Universal Robots URScript: UR10-test.urscript

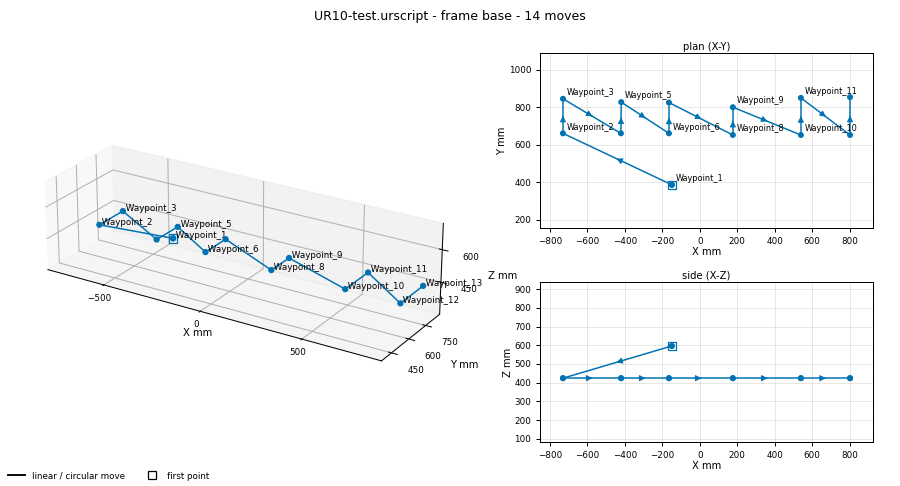
[picture p0: tool path of UR10-test.urscript in frame base, 14 of 14 moves have a stored position in this frame; points joined in program order, loops and branches not executed]
global Waypoint_1_p=p[-.148623716255, .387020693657, .596263904947, 2.224016818754, -2.218863100459, .000000000047]
global Waypoint_1_q=[-1.6361330038861635, -2.1105279423675096, 2.098508978739188, -1.5587831056934593, -1.5658103921715565, 1.5027728108834797]
global Waypoint_2_p=p[-.729817873873, .661722231264, .424287796426, -2.218887695886, 2.218882381559, -.005675531927]
global Waypoint_2_q=[-0.9138925478017441, -1.0490834600145664, 1.3516796273042528, -1.8702687876866584, -1.569889898709345, 2.2296846505934624]
global Waypoint_3_p=p[-.729817873828, .846264544764, .424287796402, -2.218887695886, 2.218882381560, -.005675531928]
global Waypoint_3_q=[-1.0153653607439015, -0.8157632596228916, 0.9656489876250722, -1.7179844037908198, -1.5701368644487452, 2.1274887333166923]
global Waypoint_4_p=p[-.420560802575, .661722231064, .424287796370, -2.218887695885, 2.218882381559, -.005675531928]
global Waypoint_4_q=[-1.2279537001817111, -1.3629806130695812, 1.794165965681119, -2.0002576570402937, -1.5708128857489623, 1.9161374014142538]
global Waypoint_5_p=p[-.418875864551, .828377650801, .424287796356, -2.218887695885, 2.218882381559, -.005675531928]
global Waypoint_5_q=[-1.2908790378613233, -1.1397118299440727, 1.489741921074341, -1.9194085745795313, -1.5708031426775904, 1.8529114400786177]
global Waypoint_6_p=p[-.164110914671, .661722231020, .424287796367, -2.218887695885, 2.218882381559, -.005675531929]
global Waypoint_6_q=[-1.5850637794811266, -1.5267522206750428, 1.9827905031090738, -2.026900558052507, -1.5711626782692507, 1.5590634072767182]
global Waypoint_7_p=p[-.164110914672, .826173042611, .424287796333, -2.218887695885, 2.218882381559, -.005675531929]
global Waypoint_7_q=[-1.582343695273308, -1.2729320930252044, 1.678075854753021, -1.9759921143142556, -1.5710752378853288, 1.5616684247757715]
global Waypoint_8_p=p[.177031398866, .652910761193, .424287796275, -2.218887695885, 2.218882381559, -.005675531929]
global Waypoint_8_q=[-2.0951142953865762, -1.535769708009413, 1.9928181636409832, -2.030398815561191, -1.5704868658568802, 1.049019558354602]
global Waypoint_9_p=p[.177031398835, .801253074719, .424287796241, -2.218887695885, 2.218882381559, -.005675531929]
global Waypoint_9_q=[-2.0015173847793495, -1.306690370177332, 1.7232682354739524, -1.9895026104403168, -1.5706322771175376, 1.1425409229913175]
global Waypoint_10_p=p[.540139343172, .652910760996, .424287796193, -2.218887695885, 2.218882381559, -.005675531929]
global Waypoint_10_q=[-2.4686027585240176, -1.2655837432115984, 1.6690811447534415, -1.9782898517891594, -1.5691603256432396, 0.6754183849426623]
global Waypoint_11_p=p[.540139343077, .850906857836, .424287796146, -2.218887695885, 2.218882381559, -.005675531929]
global Waypoint_11_q=[-2.3097959684459544, -1.0127563091339384, 1.2958725487434988, -1.8573528755436461, -1.5696233576586707, 0.8337160213651695]
global Waypoint_12_p=p[.802476144769, .652910760829, .424287796098, -2.218887695884, 2.218882381559, -.005675531929]
global Waypoint_12_q=[-2.6276425437473434, -0.9682333135372083, 1.2244082863896788, -1.8314235228237052, -1.5683444799255675, 0.5157509668525746]
global Waypoint_13_p=p[.802476144403, .855283233429, .424287795964, -2.218887695884, 2.218882381559, -.005675531927]
global Waypoint_13_q=[-2.473275530953313, -0.6975574395284951, 0.756230075928209, -1.6334802658419028, -1.5690071463035942, 0.6691447624290072]

movej(get_inverse_kin(Waypoint_1_p, qnear=Waypoint_1_q), a=1.3962634015954636, v=1.0471975511965976)
sleep(50.0)
movel(Waypoint_1_p, a=1.2, v=0.25)
movel(Waypoint_2_p, a=1.2, v=0.25)
movel(Waypoint_3_p, a=1.2, v=0.25)
movel(Waypoint_4_p, a=1.2, v=0.25)
movel(Waypoint_5_p, a=1.2, v=0.25)
movel(Waypoint_6_p, a=1.2, v=0.25)
movel(Waypoint_7_p, a=1.2, v=0.25)
movel(Waypoint_8_p, a=1.2, v=0.25)
movel(Waypoint_9_p, a=1.2, v=0.25)
movel(Waypoint_10_p, a=1.2, v=0.25)
movel(Waypoint_11_p, a=1.2, v=0.25)
movel(Waypoint_12_p, a=1.2, v=0.25)
movel(Waypoint_13_p, a=1.2, v=0.25)
